(* Logix 5000 project; controller Drives_Line1 1756-L72 rev 20.13; software revision 20.04; part 19 of 21 *)
(* tags used below, declared in another part *)
   Diamtest : BOOL;
   Diamtest_mm : REAL;
   Winder_DiamCalcOn : BOOL;
   Winder_JEC : REAL;
   Winder_JLossCrvSpd : REAL[21];
   Winder_JMaterial : REAL;
   Winder_LossCrvTrq_Pct : REAL[21];
   Winder_MatMass : REAL;
   Winder_MatVolume : REAL;
   Winder_MaxMass : REAL;
   Winder_MaxVolume : REAL;
   Winder_PctPerN : REAL;
   Winder_RatedTrq : REAL;
   Winder_RPMPerMPS : REAL;
   Winder_Running : BOOL;
   Winder_SpdMps_Flt : REAL;
   Winder_SpdRpm_Flt : REAL;
   zWinder_EncCounts : DINT;
   zWinder_JGainQ1Q2 : REAL;
   zWinder_JGainQ3Q4 : REAL;
   zWinder_MaxRate : REAL;
   zWinder_SpdReg_BWMax : REAL;
   zWinder_SpdReg_BWmin : REAL;
   zWinder_TenRefRate : REAL;
   zWinder_TenSpStall : REAL;
   zWinder_TrqLimMin_Pct : REAL;
   zWinder_TrqTrimLimMax_Pct : REAL;
   Bridle_04 : UDT_Bridle_3M;
   ExitConfig : UDT_Config_Zone;
   ExitCtrl : UDT_Control_Zone;
   LineSetpoints : UDT_Setpoints_Line;
   Out_Feedbacks : UDT_Fdbks;
   Out_Status : UDT_Status;
   par_winder_JAR : REAL;
   TestConfig_Winder : UDT_Config_Unwinder;
   TestSp_Winder : UDT_Setpoints_Unwinder;
   Winder : UDT_Winder;
   Winder_FB_Counts_mm : DINT;
   zPi : REAL;
(* P20_Winder, continued *)

ROUTINE R07_TenFb   (* function block diagram *)
   SHEET 1   // Torque Feedback
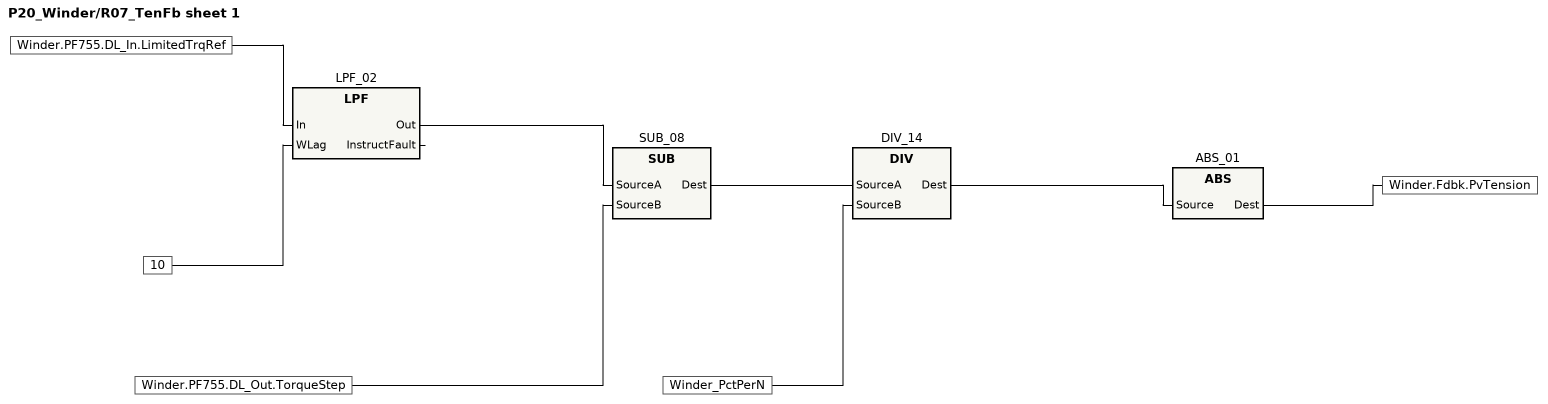
   LPF_02 : LPF(In := Winder.PF755.DL_In.LimitedTrqRef, WLag := 10);   // unwired pins: InstructFault
   SUB_08 : SUB(SourceA := LPF_02.Out, SourceB := Winder.PF755.DL_Out.TorqueStep);
   DIV_14 : DIV(SourceA := SUB_08.Dest, SourceB := Winder_PctPerN);
   ABS_01 : ABS(Source := DIV_14.Dest);
   Winder.Fdbk.PvTension := ABS_01.Dest;
   SHEET 2   // Speed Feedback
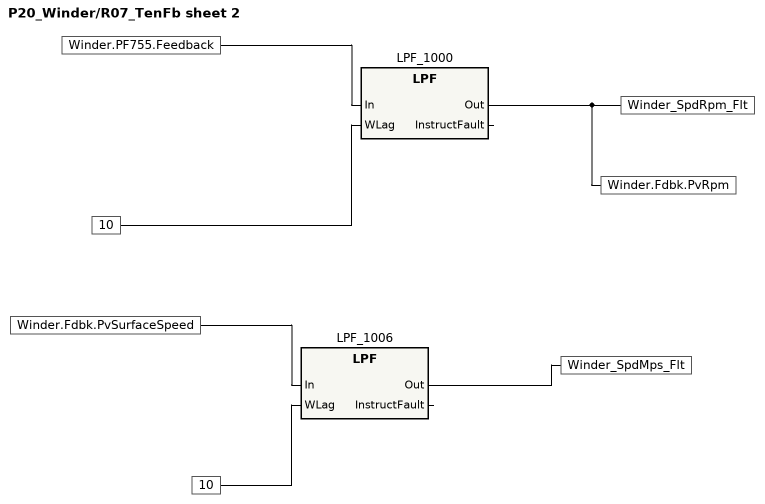
   LPF_1006 : LPF(In := Winder.Fdbk.PvSurfaceSpeed, WLag := 10);   // unwired pins: InstructFault
   LPF_1000 : LPF(In := Winder.PF755.Feedback, WLag := 10);   // unwired pins: InstructFault
   Winder_SpdMps_Flt := LPF_1006.Out;
   Winder.Fdbk.PvRpm := LPF_1000.Out;
   Winder_SpdRpm_Flt := LPF_1000.Out;
END_ROUTINE

ROUTINE R09_DiamCalc   (* function block diagram *)
   SHEET 1   // Distance/Angle Integration
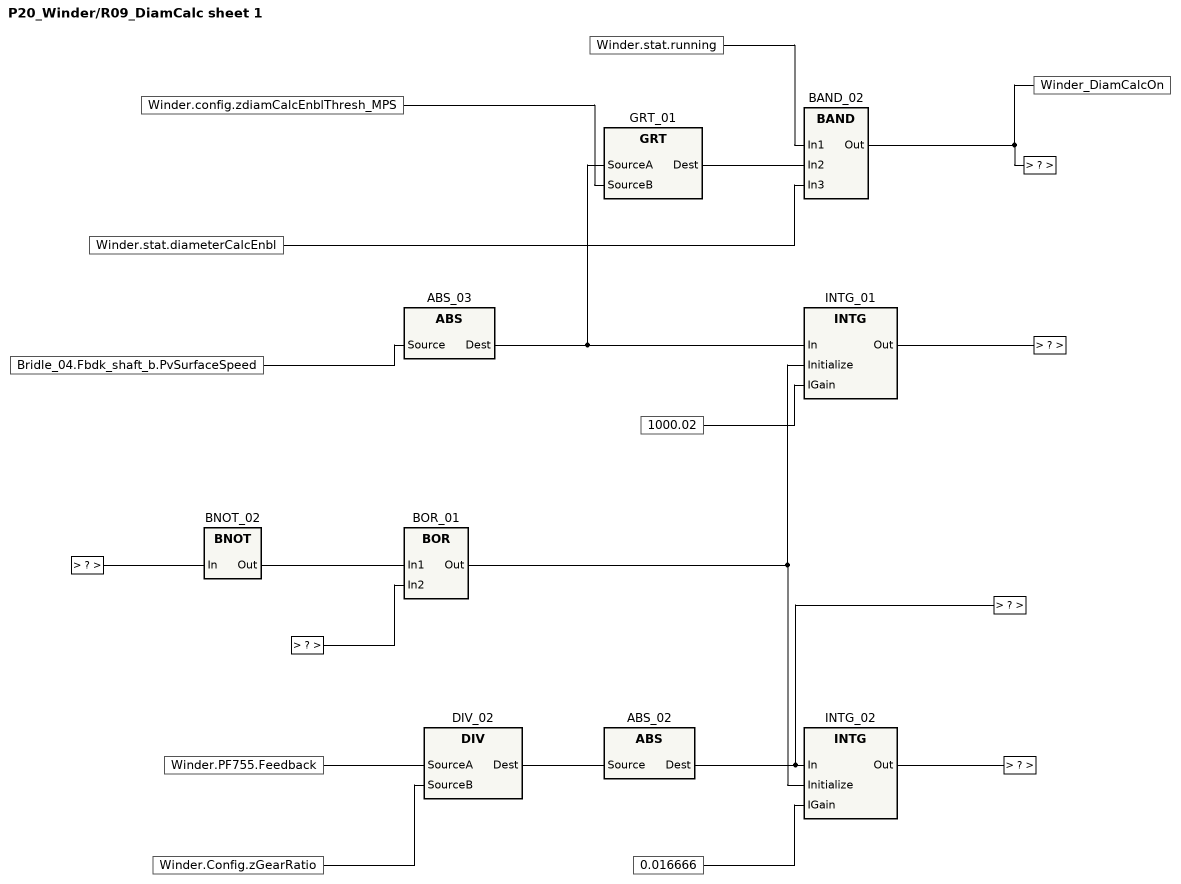
   ABS_03 : ABS(Source := Bridle_04.Fbdk_shaft_b.PvSurfaceSpeed);
   DIV_02 : DIV(SourceA := Winder.PF755.Feedback, SourceB := Winder.Config.zGearRatio);
   GRT_01 : GRT(SourceA := ABS_03.Dest, SourceB := Winder.config.zdiamCalcEnblThresh_MPS);
   ABS_02 : ABS(Source := DIV_02.Dest);
   BAND_02 : BAND(In1 := Winder.stat.running, In2 := GRT_01.Dest, In3 := Winder.stat.diameterCalcEnbl);
   WIRE(?) := ABS_02.Dest;
   BNOT_02 : BNOT(In := WIRE(?));
   BOR_01 : BOR(In1 := BNOT_02.Out, In2 := WIRE(?) {feedback});
   INTG_01 : INTG(In := ABS_03.Dest, Initialize := BOR_01.Out, IGain := 1000.02);
   INTG_02 : INTG(In := ABS_02.Dest, Initialize := BOR_01.Out, IGain := 0.016666);
   WIRE(?) := INTG_02.Out;
   WIRE(?) := BAND_02.Out;
   Winder_DiamCalcOn := BAND_02.Out;
   WIRE(?) := INTG_01.Out;
   SHEET 2   // Diameter Calculate
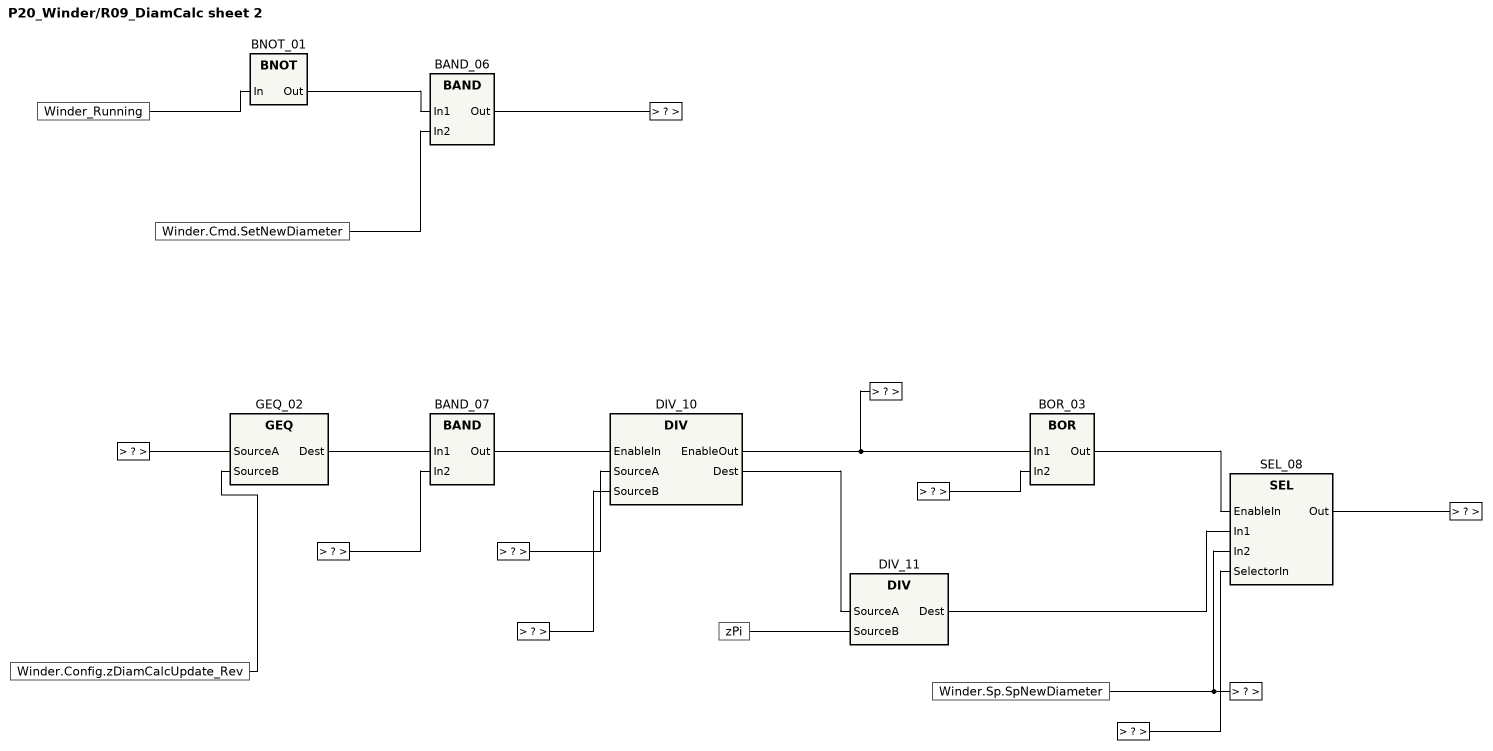
   BNOT_01 : BNOT(In := Winder_Running);
   BAND_06 : BAND(In1 := BNOT_01.Out, In2 := Winder.Cmd.SetNewDiameter);
   WIRE(?) := BAND_06.Out;
   WIRE(?) := Winder.Sp.SpNewDiameter;
   GEQ_02 : GEQ(SourceA := WIRE(?), SourceB := Winder.Config.zDiamCalcUpdate_Rev);
   BAND_07 : BAND(In1 := GEQ_02.Dest, In2 := WIRE(?));
   DIV_10 : DIV(EnableIn := BAND_07.Out, SourceA := WIRE(?), SourceB := WIRE(?));
   DIV_11 : DIV(SourceA := DIV_10.Dest, SourceB := zPi);
   WIRE(?) := DIV_10.EnableOut;
   BOR_03 : BOR(In1 := DIV_10.EnableOut, In2 := WIRE(?));
   SEL_08 : SEL(EnableIn := BOR_03.Out, In1 := DIV_11.Dest, In2 := Winder.Sp.SpNewDiameter, SelectorIn := WIRE(?));
   WIRE(?) := SEL_08.Out;
   SHEET 3   // Rate/Magnitude Limit
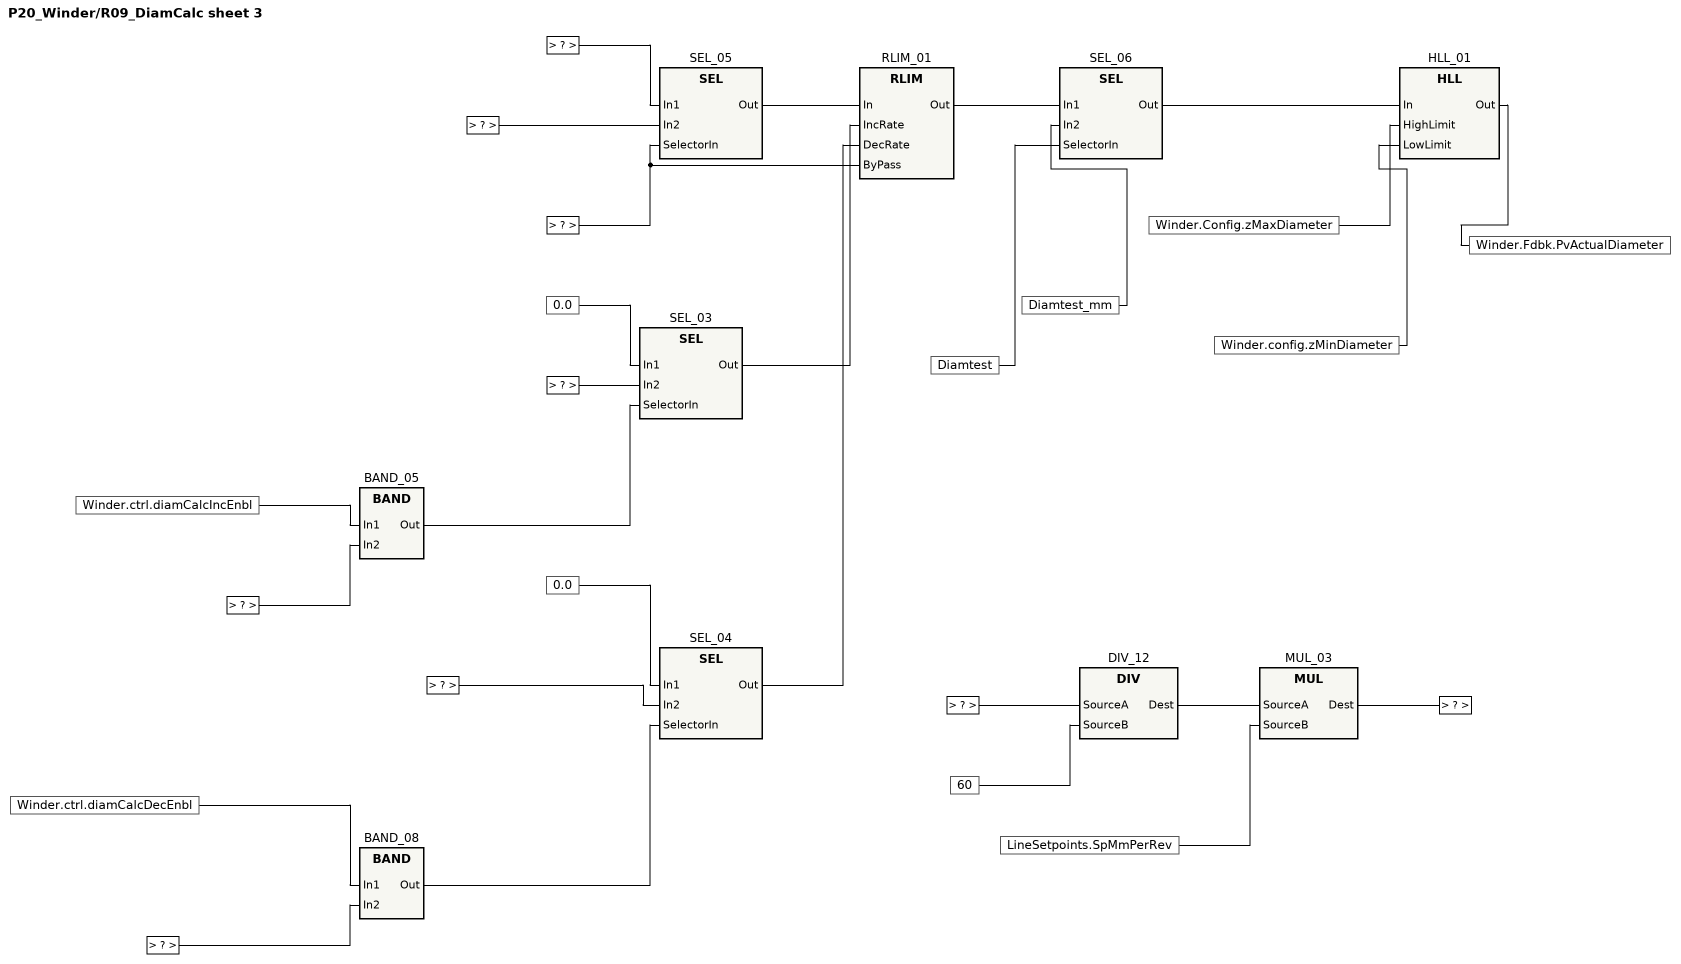
   BAND_08 : BAND(In1 := Winder.ctrl.diamCalcDecEnbl, In2 := WIRE(?));
   BAND_05 : BAND(In1 := Winder.ctrl.diamCalcIncEnbl, In2 := WIRE(?));
   SEL_04 : SEL(In1 := 0.0, In2 := WIRE(?), SelectorIn := BAND_08.Out);
   SEL_05 : SEL(In1 := WIRE(?), In2 := WIRE(?), SelectorIn := WIRE(?));
   SEL_03 : SEL(In1 := 0.0, In2 := WIRE(?), SelectorIn := BAND_05.Out);
   RLIM_01 : RLIM(In := SEL_05.Out, IncRate := SEL_03.Out, DecRate := SEL_04.Out, ByPass := WIRE(?));
   SEL_06 : SEL(In1 := RLIM_01.Out, In2 := Diamtest_mm, SelectorIn := Diamtest);
   HLL_01 : HLL(In := SEL_06.Out, HighLimit := Winder.Config.zMaxDiameter, LowLimit := Winder.config.zMinDiameter);
   Winder.Fdbk.PvActualDiameter := HLL_01.Out;
   DIV_12 : DIV(SourceA := WIRE(?), SourceB := 60);
   MUL_03 : MUL(SourceA := DIV_12.Dest, SourceB := LineSetpoints.SpMmPerRev);
   WIRE(?) := MUL_03.Dest;
END_ROUTINE

ROUTINE R10_Calculate   (* structured text *)
   // Calculate
   // Speed Conversion
   //
   // * * * * * * * * * * * * * * * * * * * * * * * * * * *
   //
   // Calculates conversion factor from surface speed [MPS] to rotational speeds [RPM].
   //
   //             Gear Ratio * 1000 [mm/M]
   // RPM/MPS =  -------------------------- * 60
   //             Roll Diameter [mm] * PI
   //
   Winder_RPMPerMPS := (Winder.Config.zGearRatio * 1000.0) / (Winder.Fdbk.PvActualDiameter * zPi) * 60;
   //
   // * * * * * * * * * * * * * * * * * * * * * * * * * * *
   //
   // Calculate
   // (Rated Motor Torque)
   //
   // * * * * * * * * * * * * * * * * * * * * * * * * * * *
   //
   //                       MtrPwrRated [KW] * 9549
   // MtrTrqRated_Nm = ----------------------------
   //                           MtrSpdBase [RPM]
   //
   Winder_RatedTrq := Winder.Config.zMotorPwr * 9549 / Winder.Config.zMtrBaseSpd;
   //
   
   
   //
   // Calculate
   // (Center Winder Inertia)
   //
   // * * * * * * * * * * * * * * * * * * * * * * * * * * *
   //
   // MaterialVolume_m3 = (Pi * (Diam_mm/2000)**2 - Pi * (DiamMinEC_mm/2000)**2) * Width_mm/1000
   //
   //Winder_MatVolume := (zPi * (Winder.Fdbk.PvActualDiameter**2) / 4)
   //- (zPi * (Winder.Config.zMinDiameter**2) / 4)* LineSetpoints.WebWidth;
   Winder_MaxVolume:= (zPi * (Winder.Config.zMaxDiameter/2000)**2)* LineSetpoints.WebWidth / 318.31;
   //
   // MaterialMass_Kg = MaterialVolume_m3 * Density_Kgm3
   //
   Winder_MatMass := Winder_MatVolume * LineSetpoints.MaterialDensity;
   Winder_MaxMass:= Winder_MaxVolume * LineSetpoints.MaterialDensity ;
   //
   // JMaterial_Kgm2 = MaterialWeight_Kg / 2 * ((Diam_mm/2000)**2 + (DiamMinEC_mm/2000)**2) / GearRatio**2
   //
   Winder_JMaterial := Winder_MatMass / 2 *
   ((Winder.Fdbk.PvActualDiameter/2000)**2 + (Winder.Config.zMinDiameter/2000)**2)
    / Winder.Config.zGearRatio**2 ;
   //
   // Calculate total reflected inertia [kilogram-meters**2]
   //
   Winder.Fdbk.PvTotalInertia := Winder_JEC + Winder_JMaterial ;
   //
   // * * * * * * * * * * * * * * * * * * * * * * * * * * *
   //
   // Calculate
   // (Normalized Inertia)
   //
   // * * * * * * * * * * * * * * * * * * * * * * * * * * *
   //
   //         J [Kgm**2] * MtrSpdBase [RPM]
   // J_Sec = -------------------------------
   //           9.549 * MtrTrqRated [Nm]
   //
   Winder.Fdbk.PvNormInertia :=
   (Winder.Fdbk.PvTotalInertia * Winder.Config.zMtrBaseSpd)
   / (9.549 * Winder_RatedTrq) ;
   
   
   (*                         Diam [mm]           100                  1      *)
   (* Conversion_PctPerN =  ----------- * -------------------- * ----------- *)
   (*                         1000 * 2       MtrTrqRated [Nm]      GearRatio  *)
   
   Winder_PctPerN := Winder.Fdbk.PvActualDiameter / Winder.Config.zGearRatio
    / Winder_RatedTrq / 20.0 ;
   
   Winder_FB_Counts_mm:= (Winder.Config.zGearRatio * zWinder_EncCounts) / (Winder.Fdbk.PvActualDiameter * zPi);
END_ROUTINE

ROUTINE R11_TenRef   (* function block diagram *)
   SHEET 1   // Tension Reference
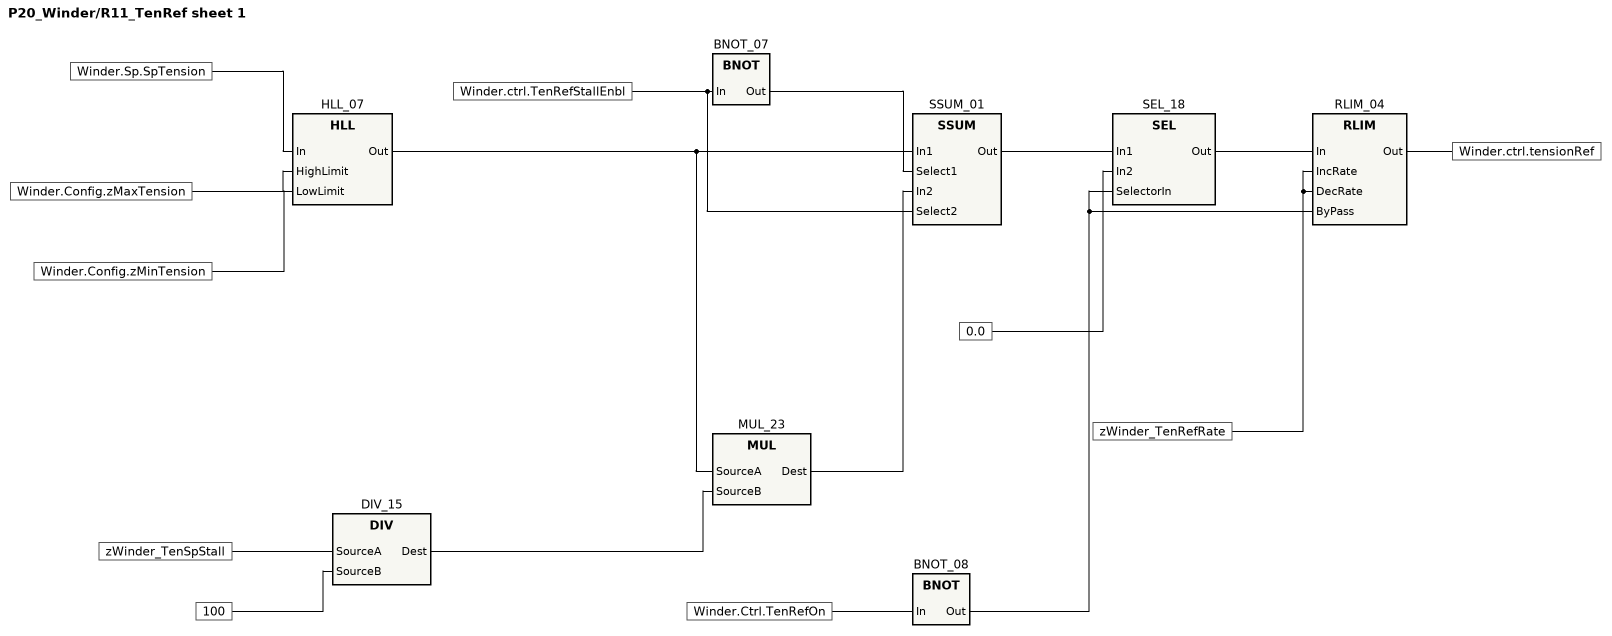
   HLL_07 : HLL(In := Winder.Sp.SpTension, HighLimit := Winder.Config.zMaxTension, LowLimit := Winder.Config.zMinTension);
   DIV_15 : DIV(SourceA := zWinder_TenSpStall, SourceB := 100);
   BNOT_07 : BNOT(In := Winder.ctrl.TenRefStallEnbl);
   MUL_23 : MUL(SourceA := HLL_07.Out, SourceB := DIV_15.Dest);
   SSUM_01 : SSUM(In1 := HLL_07.Out, Select1 := BNOT_07.Out, In2 := MUL_23.Dest, Select2 := Winder.ctrl.TenRefStallEnbl);
   BNOT_08 : BNOT(In := Winder.Ctrl.TenRefOn);
   SEL_18 : SEL(In1 := SSUM_01.Out, In2 := 0.0, SelectorIn := BNOT_08.Out);
   RLIM_04 : RLIM(In := SEL_18.Out, IncRate := zWinder_TenRefRate, DecRate := zWinder_TenRefRate, ByPass := BNOT_08.Out);
   Winder.ctrl.tensionRef := RLIM_04.Out;
END_ROUTINE

ROUTINE R12_DriveRef   (* function block diagram *)
   SHEET 1   // Select speed reference
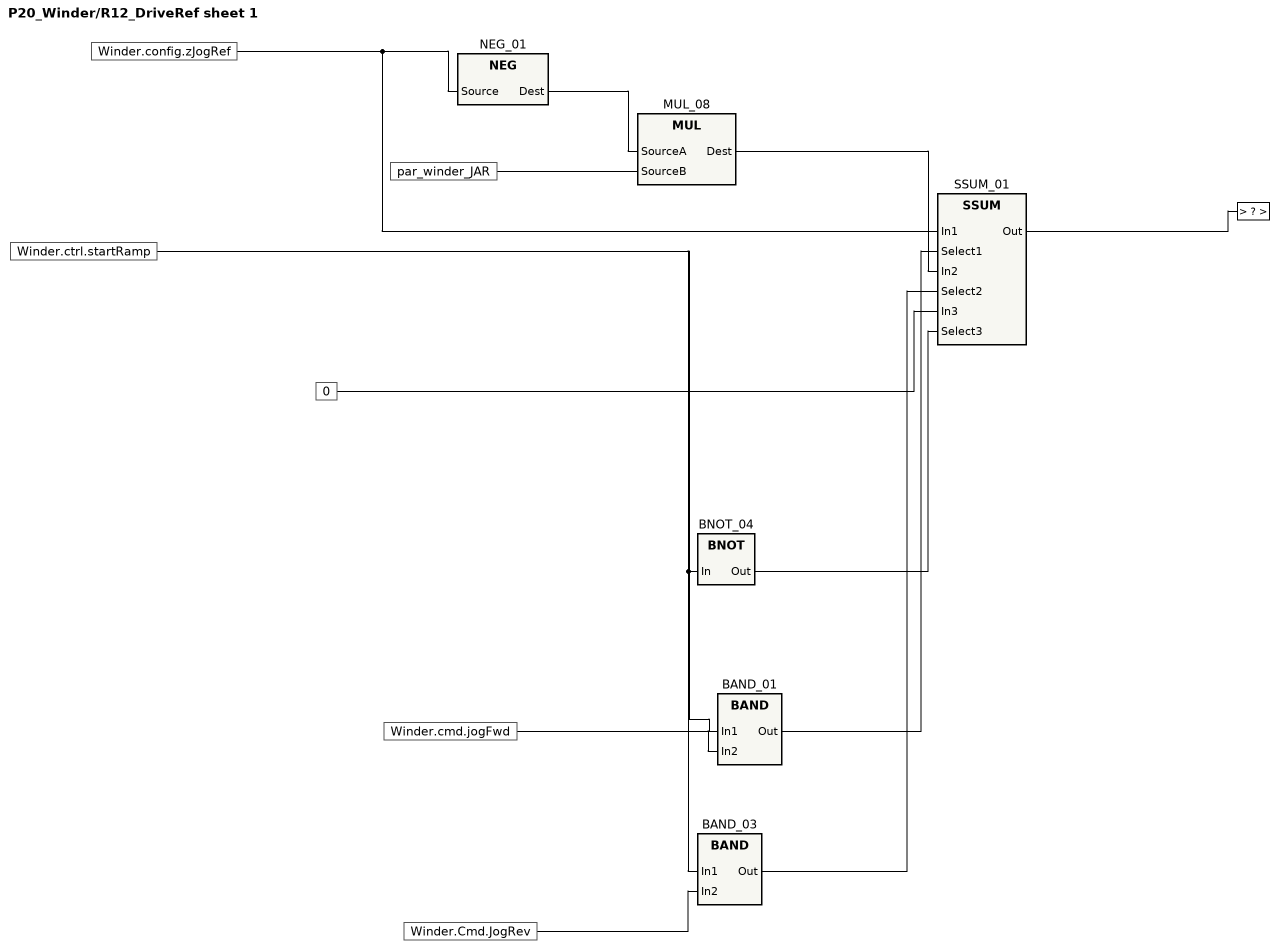
   NEG_01 : NEG(Source := Winder.config.zJogRef);
   MUL_08 : MUL(SourceA := NEG_01.Dest, SourceB := par_winder_JAR);
   BNOT_04 : BNOT(In := Winder.ctrl.startRamp);
   BAND_03 : BAND(In1 := Winder.ctrl.startRamp, In2 := Winder.Cmd.JogRev);
   BAND_01 : BAND(In1 := Winder.ctrl.startRamp, In2 := Winder.cmd.jogFwd);
   SSUM_01 : SSUM(In1 := Winder.config.zJogRef, Select1 := BAND_01.Out, In2 := MUL_08.Dest, Select2 := BAND_03.Out, In3 := 0, Select3 := BNOT_04.Out);
   WIRE(?) := SSUM_01.Out;
   SHEET 2   // S-Curve
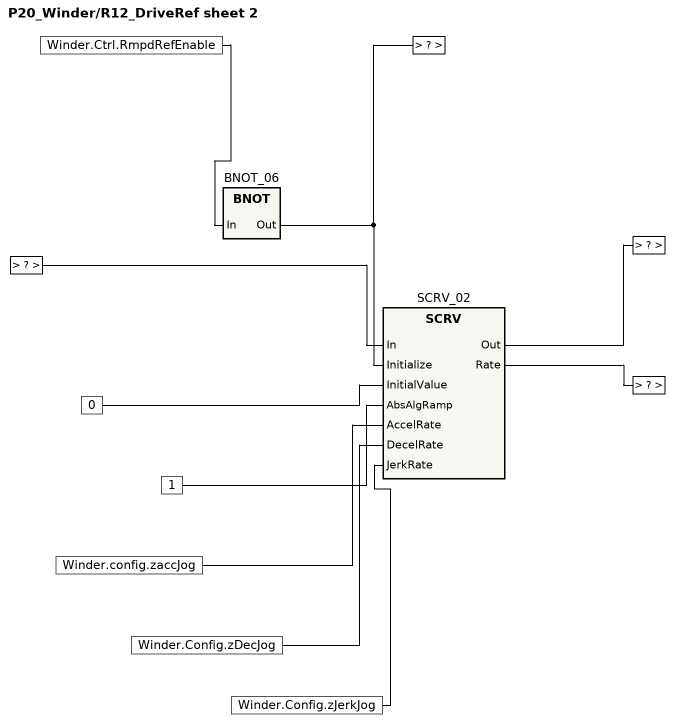
   BNOT_06 : BNOT(In := Winder.Ctrl.RmpdRefEnable);
   WIRE(?) := BNOT_06.Out;
   SCRV_02 : SCRV(In := WIRE(?), Initialize := BNOT_06.Out, InitialValue := 0, AbsAlgRamp := 1, AccelRate := Winder.config.zaccJog, DecelRate := Winder.Config.zDecJog, JerkRate := Winder.Config.zJerkJog);
   WIRE(?) := SCRV_02.Out;
   WIRE(?) := SCRV_02.Rate;
   SHEET 3   // Select ramped/unramped reference
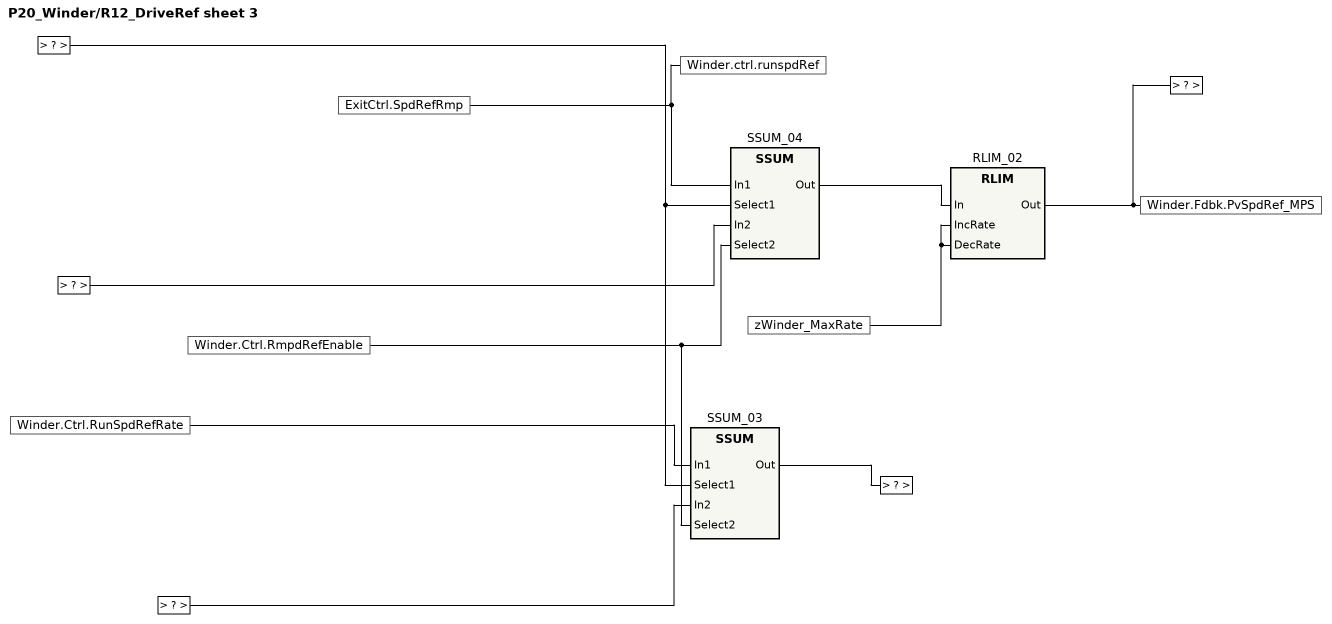
   Winder.ctrl.runspdRef := ExitCtrl.SpdRefRmp;
   SSUM_04 : SSUM(In1 := ExitCtrl.SpdRefRmp, Select1 := WIRE(?), In2 := WIRE(?), Select2 := Winder.Ctrl.RmpdRefEnable);
   RLIM_02 : RLIM(In := SSUM_04.Out, IncRate := zWinder_MaxRate, DecRate := zWinder_MaxRate);
   Winder.Fdbk.PvSpdRef_MPS := RLIM_02.Out;
   WIRE(?) := RLIM_02.Out;
   SSUM_03 : SSUM(In1 := Winder.Ctrl.RunSpdRefRate, Select1 := WIRE(?), In2 := WIRE(?), Select2 := Winder.Ctrl.RmpdRefEnable);
   WIRE(?) := SSUM_03.Out;
   SHEET 4   // Inertia Compensation
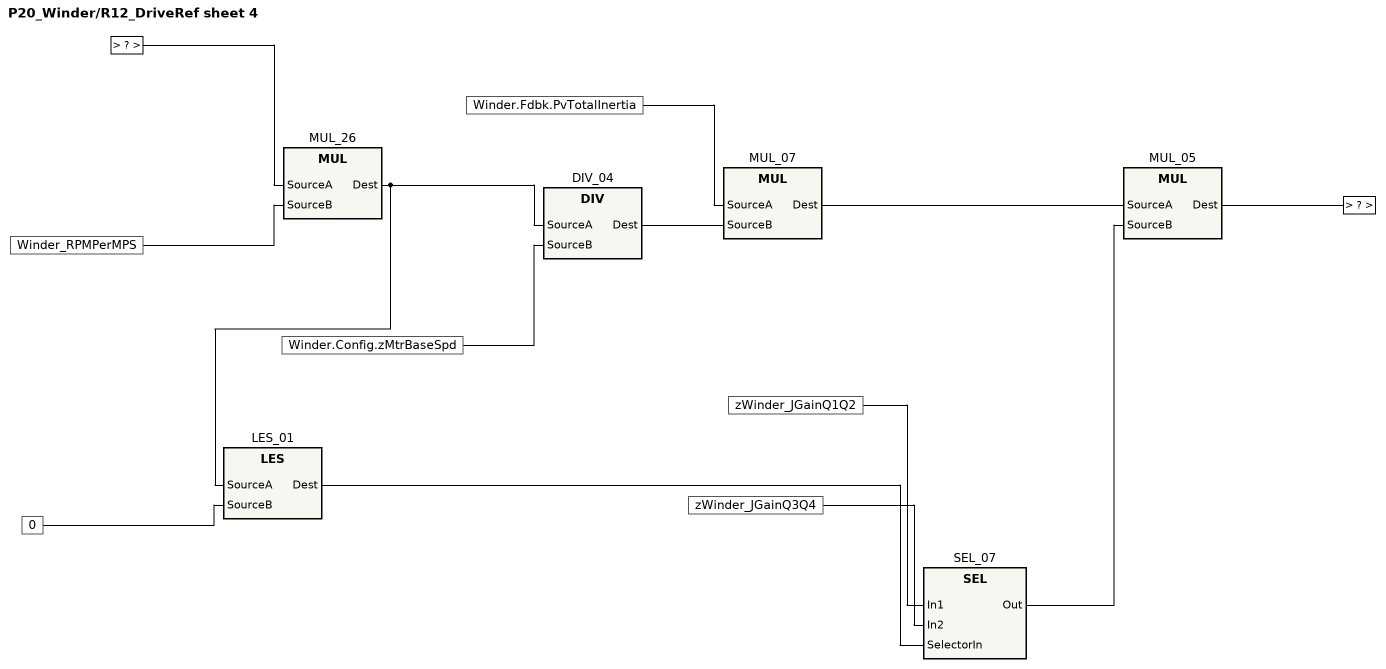
   MUL_26 : MUL(SourceA := WIRE(?), SourceB := Winder_RPMPerMPS);
   LES_01 : LES(SourceA := MUL_26.Dest, SourceB := 0);
   DIV_04 : DIV(SourceA := MUL_26.Dest, SourceB := Winder.Config.zMtrBaseSpd);
   MUL_07 : MUL(SourceA := Winder.Fdbk.PvTotalInertia, SourceB := DIV_04.Dest);
   SEL_07 : SEL(In1 := zWinder_JGainQ1Q2, In2 := zWinder_JGainQ3Q4, SelectorIn := LES_01.Dest);
   MUL_05 : MUL(SourceA := MUL_07.Dest, SourceB := SEL_07.Out);
   WIRE(?) := MUL_05.Dest;
   SHEET 5   // Friction and Windage Compensation
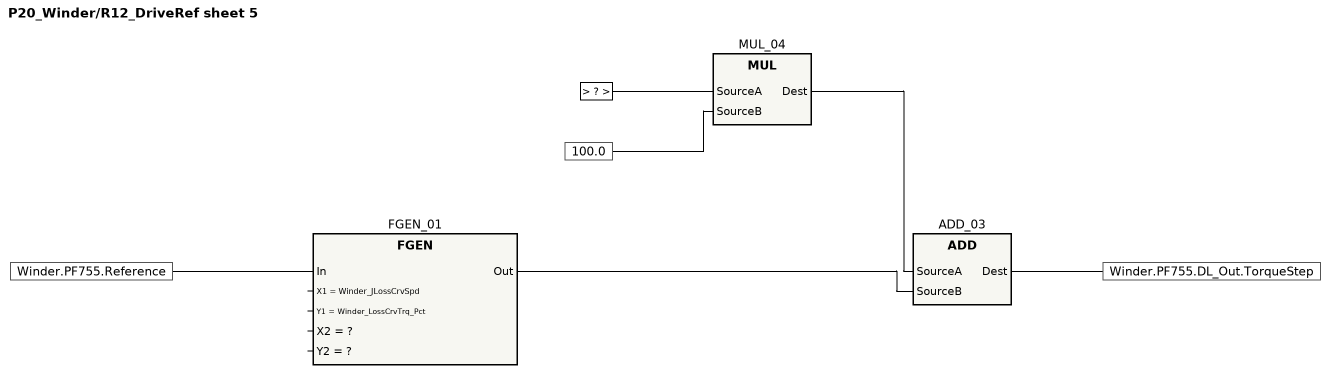
   FGEN_01 : FGEN(In := Winder.PF755.Reference, X1 := Winder_JLossCrvSpd, Y1 := Winder_LossCrvTrq_Pct, X2 := ?, Y2 := ?);
   MUL_04 : MUL(SourceA := WIRE(?), SourceB := 100.0);
   ADD_03 : ADD(SourceA := MUL_04.Dest, SourceB := FGEN_01.Out);
   Winder.PF755.DL_Out.TorqueStep := ADD_03.Dest;
   SHEET 6   // Speed trim
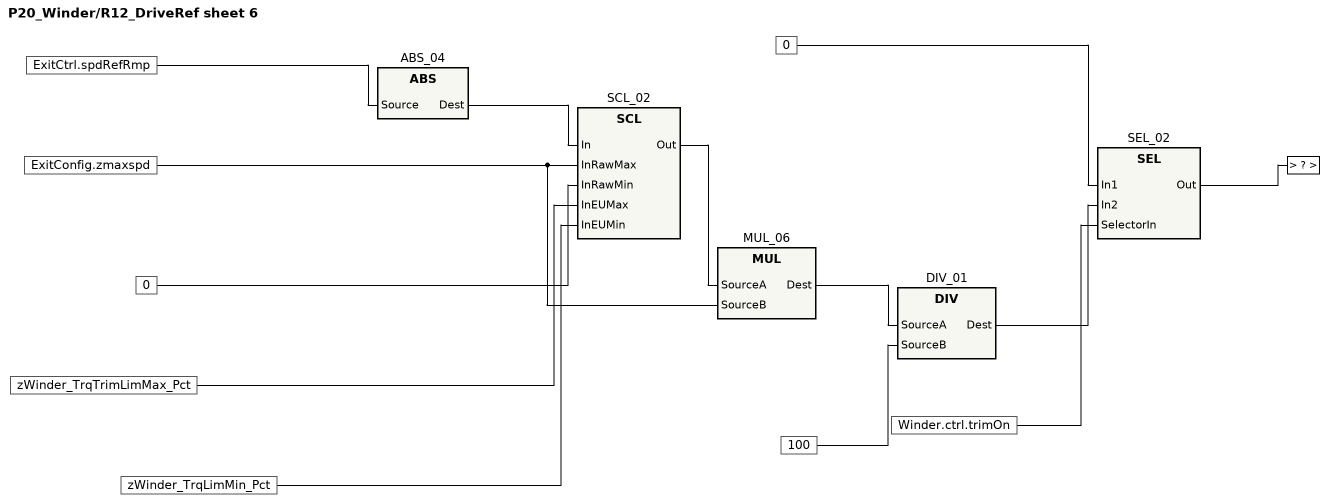
   ABS_04 : ABS(Source := ExitCtrl.spdRefRmp);
   SCL_02 : SCL(In := ABS_04.Dest, InRawMax := ExitConfig.zmaxspd, InRawMin := 0, InEUMax := zWinder_TrqTrimLimMax_Pct, InEUMin := zWinder_TrqLimMin_Pct);
   MUL_06 : MUL(SourceA := SCL_02.Out, SourceB := ExitConfig.zmaxspd);
   DIV_01 : DIV(SourceA := MUL_06.Dest, SourceB := 100);
   SEL_02 : SEL(In1 := 0, In2 := DIV_01.Dest, SelectorIn := Winder.ctrl.trimOn);
   WIRE(?) := SEL_02.Out;
   SHEET 7   // Final speed reference
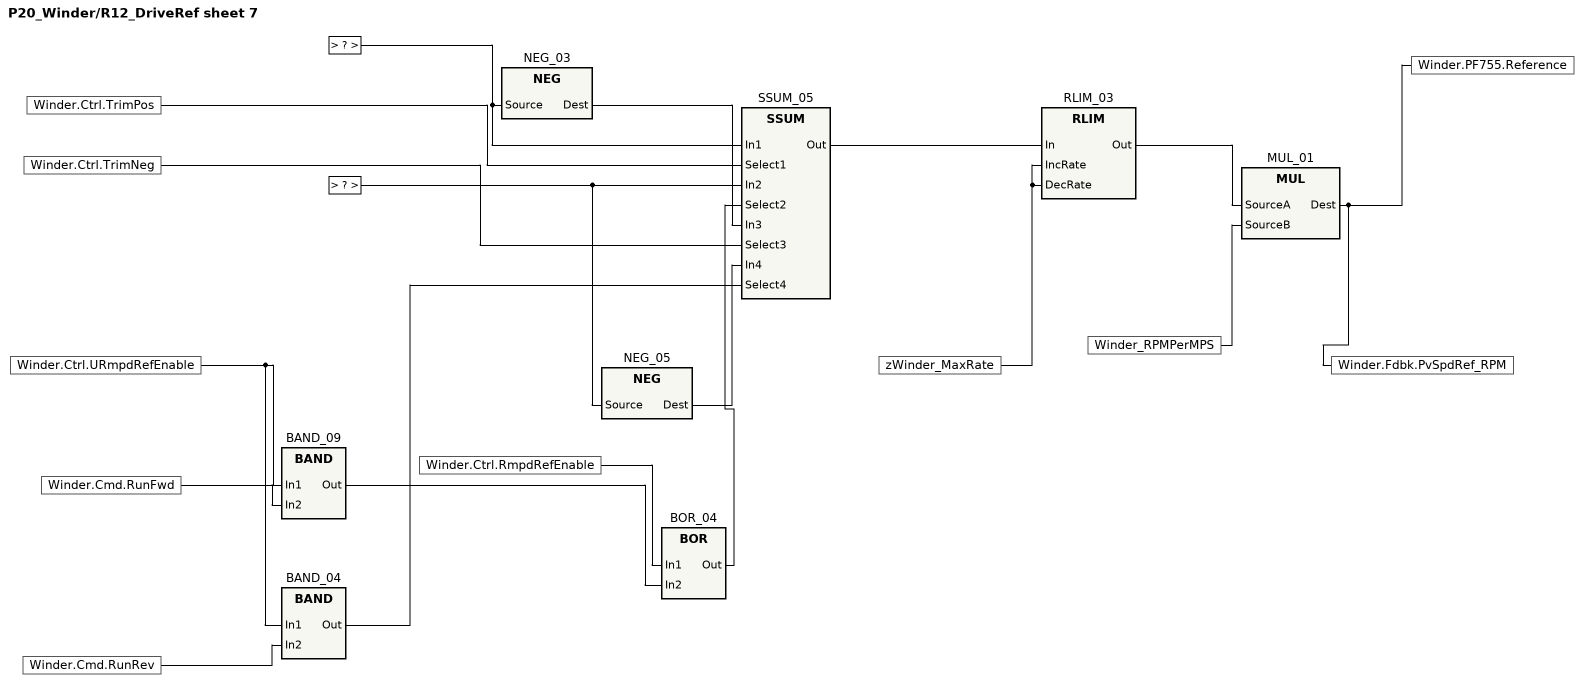
   BAND_09 : BAND(In1 := Winder.Ctrl.URmpdRefEnable, In2 := Winder.Cmd.RunFwd);
   BAND_04 : BAND(In1 := Winder.Ctrl.URmpdRefEnable, In2 := Winder.Cmd.RunRev);
   NEG_03 : NEG(Source := WIRE(?));
   NEG_05 : NEG(Source := WIRE(?));
   BOR_04 : BOR(In1 := Winder.Ctrl.RmpdRefEnable, In2 := BAND_09.Out);
   SSUM_05 : SSUM(In1 := WIRE(?), Select1 := Winder.Ctrl.TrimPos, In2 := WIRE(?), Select2 := BOR_04.Out, In3 := NEG_03.Dest, Select3 := Winder.Ctrl.TrimNeg, In4 := NEG_05.Dest, Select4 := BAND_04.Out);
   RLIM_03 : RLIM(In := SSUM_05.Out, IncRate := zWinder_MaxRate, DecRate := zWinder_MaxRate);
   MUL_01 : MUL(SourceA := RLIM_03.Out, SourceB := Winder_RPMPerMPS);
   Winder.Fdbk.PvSpdRef_RPM := MUL_01.Dest;
   Winder.PF755.Reference := MUL_01.Dest;
   SHEET 8   // Torque reference
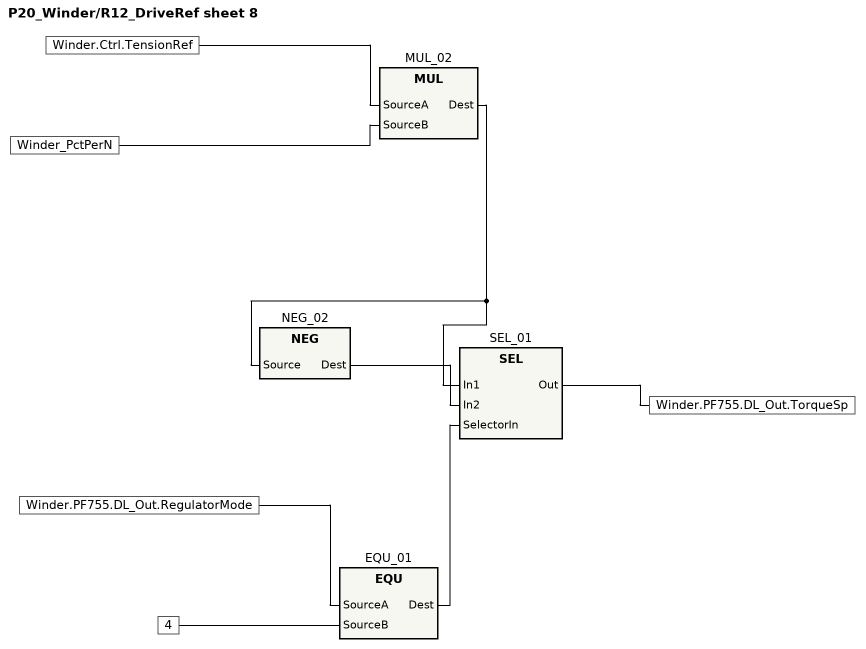
   EQU_01 : EQU(SourceA := Winder.PF755.DL_Out.RegulatorMode, SourceB := 4);
   MUL_02 : MUL(SourceA := Winder.Ctrl.TensionRef, SourceB := Winder_PctPerN);
   NEG_02 : NEG(Source := MUL_02.Dest);
   SEL_01 : SEL(In1 := MUL_02.Dest, In2 := NEG_02.Dest, SelectorIn := EQU_01.Dest);
   Winder.PF755.DL_Out.TorqueSp := SEL_01.Out;
   SHEET 9   // Speed regulator bandwidth
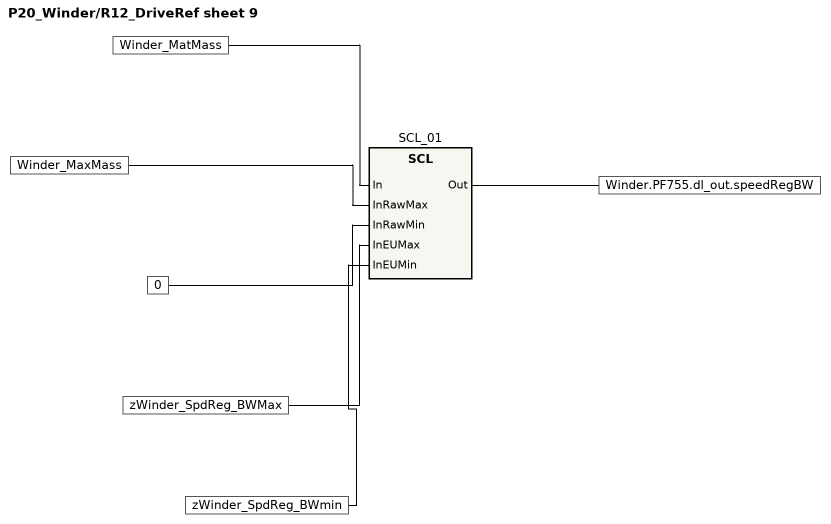
   SCL_01 : SCL(In := Winder_MatMass, InRawMax := Winder_MaxMass, InRawMin := 0, InEUMax := zWinder_SpdReg_BWMax, InEUMin := zWinder_SpdReg_BWmin);
   Winder.PF755.dl_out.speedRegBW := SCL_01.Out;
END_ROUTINE

ROUTINE R98_ToDrive   (* ladder *)
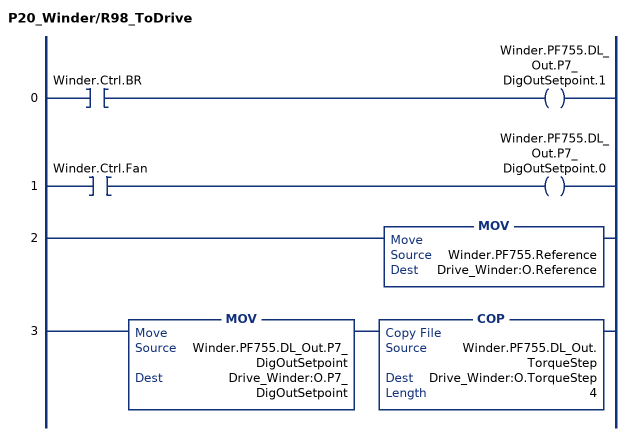
   0: XIC(Winder.Ctrl.BR)OTE(Winder.PF755.DL_Out.P7_DigOutSetpoint.1);
   1: XIC(Winder.Ctrl.Fan)OTE(Winder.PF755.DL_Out.P7_DigOutSetpoint.0);
   2: MOV(Winder.PF755.Reference,Drive_Winder:O.Reference);
   3: MOV(Winder.PF755.DL_Out.P7_DigOutSetpoint,Drive_Winder:O.P7_DigOutSetpoint)COP(Winder.PF755.DL_Out.TorqueStep,Drive_Winder:O.TorqueStep,4);
END_ROUTINE

ROUTINE R999_Test   (* ladder *)
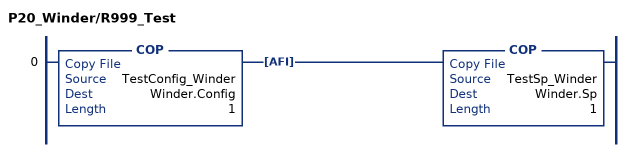
   0: COP(TestConfig_Winder,Winder.Config,1)AFI()COP(TestSp_Winder,Winder.Sp,1);
END_ROUTINE

ROUTINE R99_To_Master   (* ladder *)
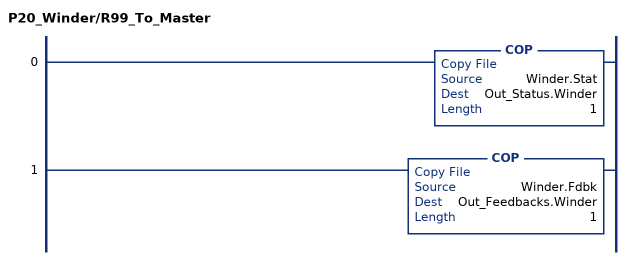
   0: COP(Winder.Stat,Out_Status.Winder,1);
   1: COP(Winder.Fdbk,Out_Feedbacks.Winder,1);
END_ROUTINE
END_PROGRAM
